PROGRAM MAIN
VAR   
 	
END_VAR

END_PROGRAM

(* stored: Version 1.1.0.1, ProductVersion 3.1.4024.12
   POU MAIN: Id {bcff7b32-2da0-4e60-839b-fea1ac037a24}, SpecialFunc None *)
